{attribute 'qualified_only'}
{attribute 'strict'}
TYPE E_PMLUnitMode :
(
	UNDEFINED		:=  0,
	AUTOMATIC		:=  1,
	MAINTENANCE 	:=  2,
	MANUAL 			:=  3,
	SEMIAUTOMATIC	:=  4,
	DRYRUN			:=  5,
	USERMODE1		:=  6,
	USERMODE2		:=  7,
	IDLE 			:=  8,
	ESTOP 			:=  9
);
END_TYPE

(* stored: Version 1.1.0.1, ProductVersion 3.1.4024.2
   DUT E_PMLUnitMode: Id {8436c567-ee42-484b-9c48-1ac6b32f7df0} *)
